TYPE DUT_1 :
STRUCT
END_STRUCT
END_TYPE

(* stored: Version 1.1.0.1, ProductVersion 3.1.4022.18
   DUT DUT_1: Id {4de0d718-9228-4bb1-b45f-807a0ed81dc7} *)
